{attribute 'qualified_only'}
{attribute 'to_string'}
TYPE MotionType :
(
	Null			:= 0,
	WaitOK			:= 1,
	Absolute		:= 2,
	Relative		:= 3,
	Time_Wait		:= 4
);
END_TYPE

(* stored: Version 1.1.0.1, ProductVersion 3.1.4026.18
   DUT MotionType: Id {6fea6617-814d-45b3-b310-af78c06a1196} *)
